// TIA Portal V19 export
FUNCTION "IPC_Manager_CALL" : Void   // FC54, LAD
TITLE = GESTIONE SCAMBIO DATI CON IPC
// stored: SetENOAutomatically false
BEGIN

REGION Network 1: Manager Call
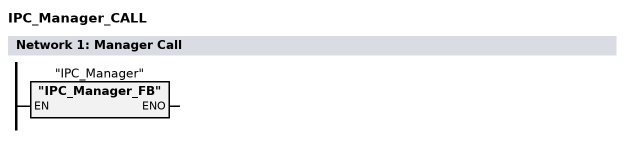
   RUNG wire#powerrail
      "IPC_Manager"()
   END_RUNG
   // the same network as SCL:
   "IPC_Manager"();   // "IPC_Manager_FB"
END_REGION
END_FUNCTION
